// TIA Portal V17 export
// export: Created 2022-12-08T10:17:24.578966Z, ExportSetting WithDefaults, DisplayName Totally Integrated Automation Portal, DisplayVersion V17 Update 5, DisplayName TIA Portal Openness, DisplayVersion V17 Update 5, DisplayName TIA Portal Version Control Interface, DisplayVersion V17, DisplayName Simotion SCOUT TIA, DisplayVersion 5.4.3.0, DisplayName SINAMICS Startdrive Advanced, DisplayVersion V17 SP1, DisplayName SINAMICS Startdrive G130, G150, S120, S150, SINAMICS MV, S210, DisplayVersion V17 SP1, DisplayName SINAMICS Startdrive G110M, G120, G120C, G120D, G120P, G115D, DisplayVersion V17 SP1, DisplayName STEP 7 Professional, DisplayVersion V17 Update 5, DisplayName STEP 7 Safety, DisplayVersion V17, DisplayName WinCC Advanced, DisplayVersion V17 Update 5
DATA_BLOCK "USER"   // DB27
{ S7_Optimized_Access := 'TRUE' }
VERSION : 0.1
// stored: AutoNumber true, DBAccessibleFromOPCUA true, DBAccessibleFromWebserver true, IsOnlyStoredInLoadMemory false, IsRetainMemResEnabled false, IsWriteProtectedInAS false, MemoryReserve 100
   VAR RETAIN
      User : Array[0.."UPPERUSERNUMBER"] of "UDT_UserManagement";
   END_VAR
BEGIN
   User[1..3].Valid := TRUE;
   User[1].UserName := 'Econo-PAK';
   User[2].UserName := 'Werkstatt';
   User[3].UserName := 'Admin';
   User[1].Password := 'EP1985';
   User[2].Password := '12345';
   User[3].Password := '123456789';
   User[1]."LogOff-Time" := 60;
   User[2]."LogOff-Time" := 10;
   User[3]."LogOff-Time" := 30;
END_DATA_BLOCK
